FUNCTION TryConvert_UINT_TO_WORD : BOOL
VAR_INPUT
	in : UINT;
	out : REFERENCE TO WORD;
END_VAR

out := UINT_TO_WORD(in);
TryConvert_UINT_TO_WORD := TRUE;

END_FUNCTION

(* stored: Version 1.1.0.1, ProductVersion 3.1.4024.12
   POU TryConvert_UINT_TO_WORD: Id {d44fcce3-7125-4fe1-945e-03fbd56342b7}, SpecialFunc None *)
